PROGRAM Case_Chase
VAR
	iState: E_MachineStates := E_MachineStates.init;
	ton1			: TON;
	ton2			: TON;
	edgepos			: R_TRIG;
	switchCounter	: UINT := 0;
END_VAR

//CASE iState OF
//	E_MachineStates.init:
//		GVL.aLights[1] := TRUE;
//		IF GVL.aSwitches[2] THEN
//			iState := E_MachineStates.pick; 
//			GVL.aLights[1] := FALSE;
//		END_IF
		
//	E_MachineStates.pick:
//		GVL.aLights[2] := TRUE;
//		IF GVL.aSwitches[3] THEN
//			iState := E_MachineStates.place;
//			GVL.aLights[2] := FALSE;
//		END_IF
		
//	E_MachineStates.place:
//		GVL.aLights[3] := TRUE;
//		IF GVL.aSwitches[4] THEN
//			iState := E_MachineStates.inspect;
//			GVL.aLights[3] := FALSE;
//		END_IF
	
//	E_MachineStates.inspect:
//	 	GVL.aLights[4] := TRUE;
//		IF GVL.aSwitches[1] THEN
//			iState := E_MachineStates.init;
//			GVL.aLights[4] := FALSE;
//		END_IF
	
//END_CASE

CASE iState OF
	
	E_MachineStates.init:
		GVL.aLights[1] := TRUE;

		// Timer 1sec switch 1
		ton1.IN := GVL.aSwitches[1];
		ton1.PT	:= T#1S;
		ton1();

		IF ton1.Q THEN
			iState := E_MachineStates.pick; 
			GVL.aLights[1] := FALSE;
		END_IF
		
	E_MachineStates.pick:
		GVL.aLights[2] := TRUE;
		
		// Counter three times on switch 2
		edgepos.CLK := gvl.aSwitches[2];
		edgepos();
		
		IF  edgepos.Q THEN
			switchCounter := switchCounter + 1;
		END_IF
		
		IF switchCounter >= 3 THEN
			iState := E_MachineStates.place;
			GVL.aLights[2]  := FALSE;
			switchCounter 	:= 0;
		END_IF
		
	E_MachineStates.place:
		GVL.aLights[3] := TRUE;
		
		// Switch 3 and 4
		IF GVL.aSwitches[3] AND GVL.aSwitches[4] THEN
			iState := E_MachineStates.inspect;
			GVL.aLights[3] := FALSE;
		END_IF
	
	E_MachineStates.inspect:
	 	GVL.aLights[4] := TRUE;
		
		// All switches off 1sec
		ton2.IN := NOT(GVL.aSwitches[1]) AND NOT(GVL.aSwitches[2]) AND NOT(GVL.aSwitches[3]) AND NOT(GVL.aSwitches[4]);
		ton2.PT := T#1S;
		ton2();
		
		IF ton2.Q THEN
			iState := E_MachineStates.init;
			GVL.aLights[4] := FALSE;
		END_IF
	
END_CASE

END_PROGRAM

(* stored: Version 1.1.0.1, ProductVersion 3.1.4024.12
   POU Case_Chase: Id {7e83de00-39e6-4566-b7d3-8ee3cda11e37}, SpecialFunc None *)
